// Mitsubishi GX Works2 project: 기계 원점 복귀   PLC: Q03UDV

PROGRAM MAIN
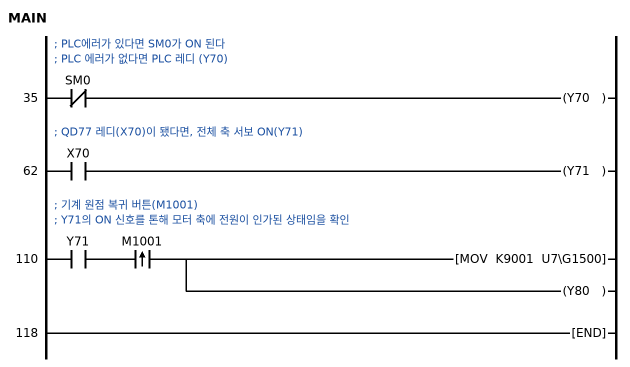
; PLC에러가 있다면 SM0가 ON 된다
; PLC 에러가 없다면 PLC 레디 (Y70)
35    LDI     SM0
      OUT     Y70
; QD77 레디(X70)이 됐다면, 전체 축 서보 ON(Y71)
62    LD      X70
      OUT     Y71
; 기계 원점 복귀 버튼(M1001)
; Y71의 ON 신호를 톤해 모터 축에 전원이 인가된 상태임을 확인
110   LD      Y71
      ANDP    M1001
      MOV     K9001 U7\G1500
      OUT     Y80
118   END
END_PROGRAM
